(*********************************** G.D S.p.A. - Technical Department ***********************************
============= PROGRAM INFO ============
FOLDER:             TBD
MACHINES INVOLVED:  TBD 

============= DESCRIPTION =============
csp main interface program

============= REVISIONS ===============
Date		Version	 	Author      	Description             
----------	-------		------------  	--------------------------------------------
2019/09/27 	0000.00	 	M.Grasso		Creation of the PRG

**********************************************************************************************************)
PROGRAM _csp_case_topRail_highest
VAR
END_VAR

csp_case_topRail();

(* CASE *)
	(* TOP RAIL *)
		(* SQUARING *)
		csp_case_topRail_squaring();

END_PROGRAM

(* stored: Version 1.1.0.1, ProductVersion 3.1.4024.3
   POU _csp_case_topRail_highest: Id {98b34573-dea7-483d-8b82-bbe10a359103}, SpecialFunc None *)
